// TIA Portal V20 export
TYPE "LER_typeCommunicationBSENDParameter"
// stored: Access Published
   STRUCT
      Input : Struct
         req : Bool;
         reset : Bool;
      END_STRUCT;
      Output : Struct
         done : Bool;
         error : Bool;
         status : Word;
      END_STRUCT;
   END_STRUCT;
END_TYPE
